FUNCTION_BLOCK SafetyMgr
VAR
  OrangeFault : BOOL;                         // Orange-level fault detected
  RedFault : BOOL;                            // Red-level fault detected
  AlarmBits : UINT;                           // Bitmask of alarmed devices
  RecoveryTrigger : BOOL;                     // Trigger for recovery attempt
  Watchdog : TON;                             // EtherCAT watchdog timer
  AllOutputsOff : BOOL;                       // All outputs are off
  ShutdownActive : ARRAY[0..19] OF BOOL;      // Shutdown in progress per device
  FastOffActive : ARRAY[0..19] OF BOOL;       // Fast off in progress per device
  AnyOutputOn : BOOL;                         // Any output is on
  EStopTimer : TON;                           // E-Stop delay timer
  RedStopTimer : TON;                         // Red Stop delay timer
  OrangeStopTimer : TON;                      // Orange Stop delay timer
  RedStopInProgress : BOOL;                   // Red stop 30s ramp is active
  OrangeStopInProgress : BOOL;                // Orange stop hold/ramp is active
  OrangeRampInProgress : BOOL;                // Orange stop 30s ramp has started (after 3min hold)
  RedStopStartTime : TIME;                    // When Red Stop ramp began
  OrangeStopStartTime : TIME;                 // When Orange Stop was first detected
  OrangeRampStartTime : TIME;                 // When Orange Stop 30s ramp began
END_VAR

// Check if a device is safe to operate
METHOD IsDeviceSafe : BOOL
VAR_INPUT
  DeviceIndex : INT;                          // Device to check
END_VAR
IsDeviceSafe := DeviceIndex >= 0 AND DeviceIndex <= 19 AND GVL.FaultLevel[DeviceIndex] = 0 AND NOT ShutdownActive[DeviceIndex];
GVL.SafetyOK[DeviceIndex] := IsDeviceSafe;    // Update safety status
END_METHOD

// Update safety conditions and system state, handling E-Stop, Red/Orange Stops, and communication faults
METHOD UpdateSafety
VAR
  devIdx : INT;            (* Device index for iteration, 0-19 *)
  anyEStop : BOOL;         (* Aggregate E-Stop state across all devices *)
  anyRedStop : BOOL;       (* Aggregate Red Stop state across all devices *)
  anyOrangeStop : BOOL;    (* Aggregate Orange Stop state across all devices *)
  systemSafe : BOOL;       (* System-wide safety condition, false if alarms active *)
  currentTime : TIME;      (* Current task time for ramp calculations *)
  elapsed_ms : DWORD;      (* Elapsed ms since stop event started *)
  rampElapsed_ms : DWORD;  (* Elapsed ms since 30s ramp phase began *)
  maintenanceMode : BOOL;  (* TRUE when GVL.SystemFlags bit 0 is set *)
END_VAR
(* Initialize aggregate safety flags *)
anyEStop := FALSE;
anyRedStop := FALSE;
anyOrangeStop := FALSE;
currentTime := TIME();

maintenanceMode := (GVL.SystemFlags AND 1) <> 0;

// Aggregate device-level safety conditions
FOR devIdx := 0 TO 19 DO
  anyEStop := anyEStop OR GVL.EStop[devIdx];         (* Check device E-Stop *)
  anyRedStop := anyRedStop OR GVL.RedStop[devIdx];   (* Check device Red Stop *)
  anyOrangeStop := anyOrangeStop OR GVL.OrangeStop[devIdx]; (* Check device Orange Stop *)
END_FOR;

// In maintenance mode, Red/Orange stops are overridden; only E-Stop applies
IF maintenanceMode THEN
  anyRedStop := FALSE;
  anyOrangeStop := FALSE;
END_IF;

// Update system state based on aggregated conditions
IF anyEStop THEN
  GVL.SystemState := 3; // E-Stop state, highest priority
ELSIF anyRedStop THEN
  GVL.SystemState := 2; // Red Stop state
ELSIF anyOrangeStop THEN
  GVL.SystemState := 1; // Orange Stop state
ELSE
  GVL.SystemState := 0; // Normal state, all clear
END_IF;

// Ramp scale: Red = 30s ramp immediately; Orange = ORANGESTOPTIME hold then 30s ramp
IF anyEStop THEN
  // E-Stop: instant off, reset all ramp state
  GVL.SystemRampScale := 0.0;
  RedStopInProgress := FALSE;
  OrangeStopInProgress := FALSE;
  OrangeRampInProgress := FALSE;
ELSIF anyRedStop THEN
  // Red Stop: 30s linear ramp-down starting immediately
  OrangeStopInProgress := FALSE;
  OrangeRampInProgress := FALSE;
  IF NOT RedStopInProgress THEN
    RedStopStartTime := currentTime;
    RedStopInProgress := TRUE;
  END_IF;
  elapsed_ms := TIME_TO_DWORD(currentTime) - TIME_TO_DWORD(RedStopStartTime);
  IF elapsed_ms >= 30000 THEN
    GVL.SystemRampScale := 0.0;
  ELSE
    GVL.SystemRampScale := 1.0 - (DWORD_TO_REAL(elapsed_ms) / 30000.0);
  END_IF;
ELSIF anyOrangeStop THEN
  // Orange Stop: hold ORANGESTOPTIME, then 30s ramp-down
  RedStopInProgress := FALSE;
  IF NOT OrangeStopInProgress THEN
    OrangeStopStartTime := currentTime;
    OrangeStopInProgress := TRUE;
    OrangeRampInProgress := FALSE;
  END_IF;
  elapsed_ms := TIME_TO_DWORD(currentTime) - TIME_TO_DWORD(OrangeStopStartTime);
  IF elapsed_ms < TIME_TO_DWORD(GVL_Constant.ORANGESTOPTIME) THEN
    GVL.SystemRampScale := 1.0; // Hold period - no ramp yet
  ELSE
    IF NOT OrangeRampInProgress THEN
      OrangeRampStartTime := currentTime;
      OrangeRampInProgress := TRUE;
    END_IF;
    rampElapsed_ms := TIME_TO_DWORD(currentTime) - TIME_TO_DWORD(OrangeRampStartTime);
    IF rampElapsed_ms >= 30000 THEN
      GVL.SystemRampScale := 0.0;
    ELSE
      GVL.SystemRampScale := 1.0 - (DWORD_TO_REAL(rampElapsed_ms) / 30000.0);
    END_IF;
  END_IF;
ELSE
  // All clear: reset state and restore full scale
  RedStopInProgress := FALSE;
  OrangeStopInProgress := FALSE;
  OrangeRampInProgress := FALSE;
  GVL.SystemRampScale := 1.0;
END_IF;

// When ramp completes (scale=0), force outputs and operation off
FOR devIdx := 0 TO 19 DO
  IF GVL.SystemRampScale <= 0.0 THEN
    GVL.OutputOn[devIdx] := FALSE;
    GVL.OperationOn[devIdx] := FALSE;
  END_IF;
END_FOR;

// Update SafetyOK per device: safe if no E-Stop, Red, or Orange Stop
FOR devIdx := 0 TO 19 DO
  GVL.SafetyOK[devIdx] := NOT (GVL.EStop[devIdx] OR GVL.RedStop[devIdx] OR GVL.OrangeStop[devIdx]);
END_FOR;

// Check system-wide alarms for safety condition
IF GVL.AlarmStatus <> 0 THEN // Non-zero AlarmStatus indicates active alarms
  systemSafe := FALSE;
ELSE
  systemSafe := TRUE;
END_IF;

// Apply system-wide safety and device-specific faults to shutdown
FOR devIdx := 0 TO 19 DO
  GVL.SafetyShutdown[devIdx] := NOT systemSafe OR GVL.CommFault[devIdx] OR GVL.TemperatureFaultHigh[devIdx];
END_FOR;

// Disable outputs for devices in shutdown
FOR devIdx := 0 TO 19 DO
  IF GVL.SafetyShutdown[devIdx] THEN
    GVL.OutputOn[devIdx] := FALSE; // Disable output on shutdown
  END_IF;
END_FOR;

// Handle recovery: clear RecoveryPending if SafetyRecovery and device is safe
FOR devIdx := 0 TO 19 DO
  IF GVL.SafetyRecovery AND GVL.SafetyOK[devIdx] THEN
    GVL.RecoveryPending[devIdx] := FALSE;
  END_IF;
END_FOR;

// Update fault level per device based on stop conditions
FOR devIdx := 0 TO 19 DO
  IF GVL.EStop[devIdx] THEN
    GVL.FaultLevel[devIdx] := 2; // Red fault level
  ELSIF GVL.OrangeStop[devIdx] THEN
    GVL.FaultLevel[devIdx] := 1; // Orange fault level
  ELSE
    GVL.FaultLevel[devIdx] := 0; // No fault
  END_IF;
END_FOR;

// Update communication faults and polling status
FOR devIdx := 0 TO 19 DO
  GVL.CommFault[devIdx] := GVL.CommTimeouts[devIdx] > GVL_constant.MAXCOMMTIMEOUT; (* Fixed: MAXCOMMTIMEOUT *)
  GVL.PollingPaused[devIdx] := GVL.CommFault[devIdx] AND NOT GVL.DataValid[devIdx]; (* Pause polling if fault and stale *)
  GVL.RecoveryPending[devIdx] := GVL.RecoveryPending[devIdx] OR (GVL.FaultLevel[devIdx] > 0); (* Set pending if faulted *)
END_FOR;
END_METHOD

END_FUNCTION_BLOCK

(* stored: Version 1.1.0.1, ProductVersion 3.1.4024.13
   POU SafetyMgr: Id {a8a109f4-0079-4314-8edc-ba599c94dc5d}, SpecialFunc None
   Method IsDeviceSafe: Id {172d67a0-935f-43f9-b8e0-3f5c9ba247dc}
   Method UpdateSafety: Id {f08a62f7-94f4-432b-9256-12fcfb147d4b} *)
